(* PLC project Tc3_EventLogger.Unsubscribe Demo, tc3-libraries-kb TwinCAT 3.1 *)
(* stored: creationDateTime 2026-05-11T01:00:00, modificationDateTime 2026-05-11T01:00:00 *)

PROGRAM P_Demo_Unsubscribe
  VAR
    fbListener : FB_ListenerBase2;  (* listener 实例 *)
    bDoUnsubscribe : BOOL := FALSE;  (* 上升沿触发 *)
    bDoUnsubscribePrev : BOOL;  (* 边沿检测 *)
    hr : HRESULT;  (* 返回值监视 *)
  END_VAR

// =============================================================================
// 场景：模块下线前取消 listener 订阅
// 价值：规范的资源释放
// 验证：先 Subscribe；再写 bDoUnsubscribe := TRUE 触发 Unsubscribe；hr 应为 S_OK
// 验证步骤：
//   1. 右键 PLC 项目 → Import PLCopenXML → 选本文件
//   2. 引用 Tc3_EventLogger（System → References → Add library）
//   3. 编译 → 登录 → 运行；按 verify 注释里给出的在线写值操作
// =============================================================================

IF bDoUnsubscribe AND NOT bDoUnsubscribePrev THEN
    hr := fbListener.Unsubscribe();
END_IF;
bDoUnsubscribePrev := bDoUnsubscribe;
END_PROGRAM
